FUNCTION_BLOCK FB_EStop
VAR_INPUT
	bEStopRaw : BOOL; // TRUE = e=stop physically pressed
	bResetButton : BOOL; // operator reset after clearing fault
END_VAR
VAR_OUTPUT
	bFaultActive : BOOL; // latched fault state
END_VAR
VAR
	rTrigEStop : R_TRIG;
	rTrigReset : R_TRIG;
END_VAR

rtrigEstop(CLK := bEStopRaw);
rtrigReset(CLK := bResetButton);

IF rtrigEStop.Q THEN
	bFaultActive := TRUE;
END_IF

IF rtrigReset.Q AND NOT bEStopRaw THEN
	bFaultActive := FALSE;
END_IF

END_FUNCTION_BLOCK

(* stored: Version 1.1.0.1, ProductVersion 3.1.4024.16
   POU FB_EStop: Id {ed360b63-46ad-4013-b52c-7064d9cb4567}, SpecialFunc None *)
